(* CODESYS project FU_dwBitGetPart.xml

Project tree, tasks and I/O mapping:
  function FU_dwBitGetPart [ST]
*)

// FU_dwBitGetPart
//This function gets only the needed bits of a variable
// |**Version**|**Author**| **Date** |**Changes**
// | 1         | NSN      | 16-03-22 | Creation
FUNCTION FU_dwBitGetPart : DWORD
VAR_INPUT
	value			:DWORD;		//Variable to get value from
	amount			:BYTE;		//Amount of bits to change
	offset			:BYTE;		//Offset in variable to change bits at
END_VAR

FU_dwBitGetPart		:=		SHR(value,offset) AND GConstants.binaryMaskDWord[amount];

END_FUNCTION
